Staubli VAL3: io.pjx

Parameters version=s7.0 stackSize=5000 millimeterUnit=true
Data file=io.dtx
